// TIA Portal V17 export
// export: Created 2022-12-08T07:31:23.3714066Z, ExportSetting WithDefaults, DisplayName Totally Integrated Automation Portal, DisplayVersion V17 Update 5, DisplayName TIA Portal Openness, DisplayVersion V17 Update 5, DisplayName TIA Portal Version Control Interface, DisplayVersion V17, DisplayName Simotion SCOUT TIA, DisplayVersion 5.4.3.0, DisplayName SINAMICS Startdrive Advanced, DisplayVersion V17 SP1, DisplayName SINAMICS Startdrive G130, G150, S120, S150, SINAMICS MV, S210, DisplayVersion V17 SP1, DisplayName SINAMICS Startdrive G110M, G120, G120C, G120D, G120P, G115D, DisplayVersion V17 SP1, DisplayName STEP 7 Professional, DisplayVersion V17 Update 5, DisplayName STEP 7 Safety, DisplayVersion V17, DisplayName WinCC Advanced, DisplayVersion V17 Update 5
FUNCTION_BLOCK "FB_Timerswitch"   // FB103, FBD
{ S7_Optimized_Access := 'TRUE' }
AUTHOR : EconoPak GmbH
VERSION : 0.1
// stored: AutoNumber true, IsIECCheckEnabled false, IsRetainMemResEnabled false, MemoryReserve 100, SetENOAutomatically true, UDAEnableTagReadback false
   VAR_OUTPUT
      q_TimerSwitch : Bool;   // Status Zeitschaltuhr 1= Heizen 0= Absenktemperatur / Status Time Switch 1= Heating 0= Temperature lowering / Tila Aikakytkin 1= Lämmitys 0= Lämpötilan lasku / Statut Interrupteur horaire 1= chauffage 0= abaissement de la température / Status Tijdschakelaar 1= Verwarming 0= Temperatuurverlaging / Status Przełącznik czasowy 1= Ogrzewanie 0= Obniżenie temperatury / Статус Переключатель времени 1= нагрев 0= понижение температуры / Estado Interruptor de tiempo 1= Calefacción 0= Bajada de temperatura
   END_VAR
   VAR_IN_OUT
      iq_TimerSwitchHMIData : "UDT_TimerSwitch";
   END_VAR
   VAR
      inst_TimerSwitch : "LGF_TimerSwitch";
   END_VAR
BEGIN

REGION Network 1: Zeitschaltuhr
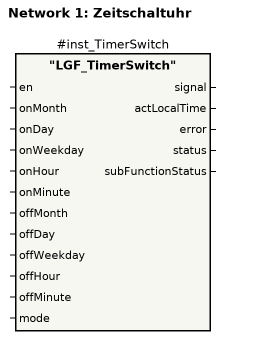
   #inst_TimerSwitch();   // "LGF_TimerSwitch"
END_REGION

REGION Network 2 (SCL): Auswahl Funktion
   CASE #iq_TimerSwitchHMIData.SelectionList OF

       2:  //Montag bis Freitag
           #inst_TimerSwitch.mode := 5;
           #inst_TimerSwitch.onHour := #iq_TimerSwitchHMIData.MoOn.HOUR;
           #inst_TimerSwitch.onMinute := #iq_TimerSwitchHMIData.MoOn.MINUTE;
           #inst_TimerSwitch.offHour := #iq_TimerSwitchHMIData.MoOff.HOUR;
           #inst_TimerSwitch.offMinute := #iq_TimerSwitchHMIData.MoOff.MINUTE;

       3:  //Montag bis Sonntag
           #inst_TimerSwitch.mode := 1;
           #inst_TimerSwitch.onHour := #iq_TimerSwitchHMIData.MoOn.HOUR;
           #inst_TimerSwitch.onMinute := #iq_TimerSwitchHMIData.MoOn.MINUTE;
           #inst_TimerSwitch.offHour := #iq_TimerSwitchHMIData.MoOff.HOUR;
           #inst_TimerSwitch.offMinute := #iq_TimerSwitchHMIData.MoOff.MINUTE;

       4:  //Wöchentlich
           #inst_TimerSwitch.mode := 2;
           #inst_TimerSwitch.onWeekday := #iq_TimerSwitchHMIData.SelectionListWeeklyOn;
           #inst_TimerSwitch.offWeekday := #iq_TimerSwitchHMIData.SelectionListWeeklyOff;
           #inst_TimerSwitch.onHour := #iq_TimerSwitchHMIData.MoOn.HOUR;
           #inst_TimerSwitch.onMinute := #iq_TimerSwitchHMIData.MoOn.MINUTE;
           #inst_TimerSwitch.offHour := #iq_TimerSwitchHMIData.MoOff.HOUR;
           #inst_TimerSwitch.offMinute := #iq_TimerSwitchHMIData.MoOff.MINUTE;

       5:  //Täglich
           #inst_TimerSwitch.mode := 1;
           CASE #inst_TimerSwitch.actLocalTime.WEEKDAY OF
               1:
                   #inst_TimerSwitch.onHour := #iq_TimerSwitchHMIData.SunOn.HOUR;
                   #inst_TimerSwitch.onMinute := #iq_TimerSwitchHMIData.SunOn.MINUTE;
                   #inst_TimerSwitch.offHour := #iq_TimerSwitchHMIData.SunOff.HOUR;
                   #inst_TimerSwitch.offMinute := #iq_TimerSwitchHMIData.SunOff.MINUTE;

               2:
                   #inst_TimerSwitch.onHour := #iq_TimerSwitchHMIData.MoOn.HOUR;
                   #inst_TimerSwitch.onMinute := #iq_TimerSwitchHMIData.MoOn.MINUTE;
                   #inst_TimerSwitch.offHour := #iq_TimerSwitchHMIData.MoOff.HOUR;
                   #inst_TimerSwitch.offMinute := #iq_TimerSwitchHMIData.MoOff.MINUTE;

               3:
                   #inst_TimerSwitch.onHour := #iq_TimerSwitchHMIData.TuesOn.HOUR;
                   #inst_TimerSwitch.onMinute := #iq_TimerSwitchHMIData.TuesOn.MINUTE;
                   #inst_TimerSwitch.offHour := #iq_TimerSwitchHMIData.TuesOff.HOUR;
                   #inst_TimerSwitch.offMinute := #iq_TimerSwitchHMIData.TuesOff.MINUTE;

               4:
                   #inst_TimerSwitch.onHour := #iq_TimerSwitchHMIData.WedOn.HOUR;
                   #inst_TimerSwitch.onMinute := #iq_TimerSwitchHMIData.WedOn.MINUTE;
                   #inst_TimerSwitch.offHour := #iq_TimerSwitchHMIData.WedOff.HOUR;
                   #inst_TimerSwitch.offMinute := #iq_TimerSwitchHMIData.WedOff.MINUTE;

               5:
                   #inst_TimerSwitch.onHour := #iq_TimerSwitchHMIData.ThursOn.HOUR;
                   #inst_TimerSwitch.onMinute := #iq_TimerSwitchHMIData.ThursOn.MINUTE;
                   #inst_TimerSwitch.offHour := #iq_TimerSwitchHMIData.ThursOff.HOUR;
                   #inst_TimerSwitch.offMinute := #iq_TimerSwitchHMIData.ThursOff.MINUTE;

               6:
                   #inst_TimerSwitch.onHour := #iq_TimerSwitchHMIData.FriOn.HOUR;
                   #inst_TimerSwitch.onMinute := #iq_TimerSwitchHMIData.FriOn.MINUTE;
                   #inst_TimerSwitch.offHour := #iq_TimerSwitchHMIData.FriOff.HOUR;
                   #inst_TimerSwitch.offMinute := #iq_TimerSwitchHMIData.FriOff.MINUTE;

               7:
                   #inst_TimerSwitch.onHour := #iq_TimerSwitchHMIData.SatOn.HOUR;
                   #inst_TimerSwitch.onMinute := #iq_TimerSwitchHMIData.SatOn.MINUTE;
                   #inst_TimerSwitch.offHour := #iq_TimerSwitchHMIData.SatOff.HOUR;
                   #inst_TimerSwitch.offMinute := #iq_TimerSwitchHMIData.SatOff.MINUTE;
           END_CASE;
   END_CASE;
END_REGION

REGION Network 3 (SCL): Ansteuerung Ausgang Zeitschaltuhr
   IF #iq_TimerSwitchHMIData.SelectionList <= 1
   THEN
       #q_TimerSwitch := #iq_TimerSwitchHMIData.SelectionList.%X0;
   ELSE
       #q_TimerSwitch := #inst_TimerSwitch.signal;
   END_IF;
END_REGION
END_FUNCTION_BLOCK
